{attribute 'linkalways'} 
{attribute 'no_explicit_call' := 'This FB is a CLASS and must be accessed using methods or properties'}
{attribute 'enable_dynamic_creation'}
FUNCTION_BLOCK FINAL NOT_USINT EXTENDS Node
VAR
	in : _USINT(0);
	out : _USINT(0);
END_VAR

METHOD PUBLIC Clone : I_Node
VAR
	pNode : POINTER TO NOT_USINT;
END_VAR
pNode := __NEW(NOT_USINT);
Clone := pNode^;
END_METHOD

METHOD FB_init : BOOL
VAR_INPUT
	bInitRetains : BOOL; // if TRUE, the retain variables are initialized (warm start / cold start)
	bInCopyCode : BOOL;  // if TRUE, the instance afterwards gets moved into the copy code (online change)
END_VAR
AddInput('in',THIS^.in);
AddOutput('out', THIS^.out);
END_METHOD

METHOD PROTECTED OnExecute
VAR
END_VAR
out.Value := NOT in.Value;
END_METHOD

END_FUNCTION_BLOCK

(* stored: Version 1.1.0.1, ProductVersion 3.1.4024.15
   POU NOT_USINT: Id {9aebc583-a0b1-43ef-80f2-a43d5cd9134c}, SpecialFunc None
   Folder Constructor: Id {c820b9f5-bee8-4726-8a1b-9d52fd89a279}
   Method Clone: Id {84b55d78-a362-4481-ac7d-d33b68daf5a6}
   Method FB_init: Id {cc6c5c80-017d-4195-9ac2-544c9ea4ba8e}
   Method OnExecute: Id {fcd339e1-b5f5-4efe-b269-4e3ecb4bb409} *)
